INTERFACE IBase EXTENDS __System.IQueryInterface

END_INTERFACE

(* stored: Version 1.1.0.1, ProductVersion 3.1.4024.12
   Itf IBase: Id {694937b0-3980-4bb3-9842-90b0a3f65fbe} *)
